// TIA Portal V17 export
// export: Created 2023-06-23T18:33:41.1596707Z, ExportSetting WithDefaults, DisplayName Totally Integrated Automation Portal, DisplayVersion V17, DisplayName TIA Portal Openness, DisplayVersion V17, DisplayName TIA Portal Version Control Interface, DisplayVersion V17, DisplayName STEP 7 Professional, DisplayVersion V17, DisplayName STEP 7 Safety, DisplayVersion V17, DisplayName WinCC Advanced / Unified PC, DisplayVersion V17
VAR_GLOBAL   // PLC tag table "27_ELR-2"
   "iELR-2" AT %I13.4 : Bool;
   "oELR-2" AT %Q12.7 : Bool;
END_VAR
